FUNCTION_BLOCK F_LWORD_TO_STRING (* convert LWORD to STRING *)
  (* Standard: 61131-3; Classification: type conversion function *)
  (* Version 0.0, 2012-01-18, 4DIAC-IDE, 4DIAC-Consortium *)
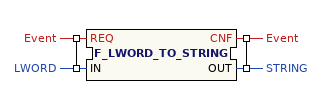
  EVENT_INPUT
    REQ WITH IN; (* Service Request *)
  END_EVENT
  EVENT_OUTPUT
    CNF WITH OUT; (* Confirmation of Requested Service *)
  END_EVENT
  VAR_INPUT
    IN : LWORD; (* Event Input Qualifier *)
  END_VAR
  VAR_OUTPUT
    OUT : STRING; (* Event Output Qualifier *)
  END_VAR
END_FUNCTION_BLOCK
